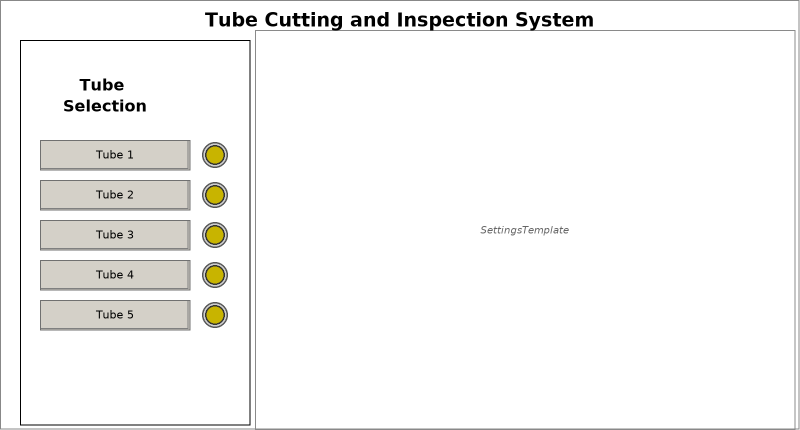
VISUALIZATION Settings  // 800x430
    Frame (255,30 540x400)
        shows SettingsTemplate(Tube := MAIN.TubeHmi)
        shows SettingsTemplate(Tube := MAIN.TubeSelection[2])
        shows SettingsTemplate(Tube := MAIN.TubeSelection[3])
        shows SettingsTemplate(Tube := MAIN.TubeSelection[4])
        shows SettingsTemplate(Tube := MAIN.TubeSelection[5])
    Label (10,79 170x30)
    Label (0,5 800x30), "Tube Cutting and Inspection System"
    Group (20,65 230x51)
        Label (0,21 170x30), "Selection"
        Label (0,0 170x30), "Tube"
    Rectangle (20,40 230x385)
    Button (40,140 150x30), "Tube 1"
        OnMouseClick: execute {
            MAIN.TubeHmi := MAIN.TubeSelection[1];
            MAIN.TubeIndicator[1] := TRUE;
            MAIN.TubeIndicator[2] := FALSE;
            MAIN.TubeIndicator[3] := FALSE;
            MAIN.TubeIndicator[4] := FALSE;
            MAIN.TubeIndicator[5] := FALSE;
        }
    Button (40,180 150x30), "Tube 2"
        OnMouseClick: execute {
            MAIN.TubeHmi := MAIN.TubeSelection[2];
            MAIN.TubeIndicator[1] := FALSE;
            MAIN.TubeIndicator[2] := TRUE;
            MAIN.TubeIndicator[3] := FALSE;
            MAIN.TubeIndicator[4] := FALSE;
            MAIN.TubeIndicator[5] := FALSE;
        }
    Button (40,220 150x30), "Tube 3"
        OnMouseClick: execute {
            MAIN.TubeHmi := MAIN.TubeSelection[3];
            MAIN.TubeIndicator[1] := FALSE;
            MAIN.TubeIndicator[2] := FALSE;
            MAIN.TubeIndicator[3] := TRUE;
            MAIN.TubeIndicator[4] := FALSE;
            MAIN.TubeIndicator[5] := FALSE;
        }
    Button (40,260 150x30), "Tube 4"
        OnMouseClick: execute {
            Main.TubeHmi := MAIN.TubeSelection[4];
            MAIN.TubeIndicator[1] := FALSE;
            MAIN.TubeIndicator[2] := FALSE;
            MAIN.TubeIndicator[3] := FALSE;
            MAIN.TubeIndicator[4] := TRUE;
            MAIN.TubeIndicator[5] := FALSE;
        }
    Button (40,300 150x30), "Tube 5"
        OnMouseClick: execute {
            Main.TubeHmi := MAIN.TubeSelection[5];
            MAIN.TubeIndicator[1] := FALSE;
            MAIN.TubeIndicator[2] := FALSE;
            MAIN.TubeIndicator[3] := FALSE;
            MAIN.TubeIndicator[4] := FALSE;
            MAIN.TubeIndicator[5] := TRUE;
        }
    Lamp1 (200,140 30x30), variable: MAIN.TubeIndicator[1], style: Lamp-Lamp1-Yellow
    Lamp1 (200,180 30x30), variable: MAIN.TubeIndicator[2], style: Lamp-Lamp1-Yellow
    Lamp1 (200,220 30x30), variable: MAIN.TubeIndicator[3], style: Lamp-Lamp1-Yellow
    Lamp1 (200,260 30x30), variable: MAIN.TubeIndicator[4], style: Lamp-Lamp1-Yellow
    Lamp1 (200,300 30x30), variable: MAIN.TubeIndicator[5], style: Lamp-Lamp1-Yellow
    Group (20,70 230x51)
        Label (0,21 170x30), "Selection"
        Label (0,0 170x30), "Tube"
END_VISUALIZATION

(* stored: Version 1.1.0.1, ProductVersion 3.1.4024.3
   Visu Settings: Id {c425db74-4fc6-4531-abcd-3ec6e8aff5a3} *)
